Staubli VAL3: start.pgx

program start()
begin
  call init()

  while (bBLOQ_CTRL==false)
    call Comunicacion()
    call JOGG_PC()
    delay(0)
  endWhile

end
